FUNCTION_BLOCK FB_LGHeatpump implements IF_Heatpump
VAR_IN_OUT
	MBMaster		:	ModbusRtuMasterV2_KL6x22B;
END_VAR

VAR_OUTPUT
	Get				:	ST_HeatPump_Get;

END_VAR

VAR_IN_OUT CONSTANT
	st_params		: 	ST_Coolingsystem_params;
END_VAR

VAR_INPUT
	ACPowerStatus	:	BOOL;
	HeatPumpID		:	BYTE;
	SFCInit			:	BOOL;
	e_ID				:	eObject_ID := eObject_ID.HeatPump;
END_VAR
		
VAR
	ton_MBBUSYTimeOut		: TON := (PT := T#10s);
	DataBuffer				:	ARRAY[0..50] OF WORD;
	ton_modbusStuckTrigger	:	Ton	:=	(PT := T#5S);
	Ton_ErrorTimer			:	Ton := (PT := T#5M);
	MBRetryCount			:	BYTE;
	MBFree					:	BOOL;
	bMBActive				:	BOOL;
	ftrig_ModbusStartTrigger		:	f_Trig;
	TransmissionDoneTrigger	:	F_Trig;
	rtrig_ManualModbusStartTrigger : r_trig;
	btest	:	BOOL;
	ManADDR : BYTE;
	ton_testTimer	:	Ton := (Pt := T#100MS);
	TP_ModbusStartTriggerDelay	:	TP := (PT := TIME#50MS);
	u_counter				:	UINT;
END_VAR

VAR
	RequestedSetpoint				:	st_OperatingPoint;
	b_EMStop						:	BOOL;
	b_resetErrors					:	BOOL;
	t_RemainingPreheatingTime	:	TIME;
	sPressureErrorText			:	STRING;
	sCompressorErrorText		:	STRING;
	sPumpErrorText				:	STRING;
	sWaterTempErrorText			:	STRING;
END_VAR

VAR PERSISTENT
	dt_LastHPOperationTime	:	DT := DT#1970-1-1-0:0:0.000;
END_VAR


VAR
	CoilStatus		:	BYTE;
	LGget	:	LG_get;
	LGset	:	LG_SET;

	HeatpumpEMOperationAvailable	:	Bool;
END_VAR

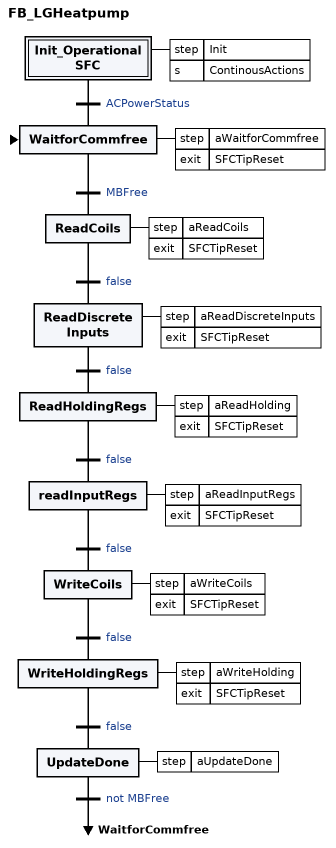
INITIAL_STEP Init_OperationalSFC:
    Init(N);  // step action
    ContinousActions(s);
END_STEP
TRANSITION FROM Init_OperationalSFC TO WaitforCommfree
    := ACPowerStatus;
END_TRANSITION
STEP WaitforCommfree:
    aWaitforCommfree(N);  // step action
    SFCTipReset(P0);  // exit action
END_STEP
TRANSITION FROM WaitforCommfree TO ReadCoils
    := MBFree;
END_TRANSITION
STEP ReadCoils:  // max time T#2S
    aReadCoils(N);  // step action
    SFCTipReset(P0);  // exit action
END_STEP
TRANSITION FROM ReadCoils TO ReadDiscreteInputs
    := false;
END_TRANSITION
STEP ReadDiscreteInputs:
    aReadDiscreteInputs(N);  // step action
    SFCTipReset(P0);  // exit action
END_STEP
TRANSITION FROM ReadDiscreteInputs TO ReadHoldingRegs
    := false;
END_TRANSITION
STEP ReadHoldingRegs:
    aReadHolding(N);  // step action
    SFCTipReset(P0);  // exit action
END_STEP
TRANSITION FROM ReadHoldingRegs TO readInputRegs
    := false;
END_TRANSITION
STEP readInputRegs:
    aReadInputRegs(N);  // step action
    SFCTipReset(P0);  // exit action
END_STEP
TRANSITION FROM readInputRegs TO WriteCoils
    := false;
END_TRANSITION
STEP WriteCoils:
    aWriteCoils(N);  // step action
    SFCTipReset(P0);  // exit action
END_STEP
TRANSITION FROM WriteCoils TO WriteHoldingRegs
    := false;
END_TRANSITION
STEP WriteHoldingRegs:
    aWriteHolding(N);  // step action
    SFCTipReset(P0);  // exit action
END_STEP
TRANSITION FROM WriteHoldingRegs TO UpdateDone
    := false;
END_TRANSITION
STEP UpdateDone:
    aUpdateDone(N);  // step action
END_STEP
TRANSITION FROM UpdateDone TO WaitforCommfree
    := not MBFree;
END_TRANSITION

METHOD AllowMBComm : BOOL
VAR_INPUT
	b_AllowComm	:	Bool;
END_VAR
MBFree	:= b_AllowComm;
END_METHOD

ACTION aReadCoils:
bMBActive := TRUE;

MBMaster.ReadCoils(	UnitID 		:= 	HeatPumpID,
					Quantity 	:= 	5,
					MBAddr		:=	0,				
					cbLength 	:= 	6,
					pMemoryAddr	:=	ADR(CoilStatus),
					Execute		:=	ftrig_ModbusStartTrigger.Q,
				);
	

IF TransmissionDoneTrigger.q THEN
	IF NOT MBMaster.Error THEN
		//Full datastruct for debug purposes. Can be removed later
		LGget.Coils.b_EnableOperation := CoilStatus.0;
		LGget.Coils.b_EnableSwwOperation := CoilStatus.1;
		LGget.Coils.b_EnableSilentMode := CoilStatus.2;
		LGget.Coils.b_EnableDesinfectionMode := Coilstatus.3;
		LGget.Coils.b_EmstopActive := CoilStatus.4;
		LGget.Coils.b_EnableEmStop := CoilStatus.5;
		//Full datastruct for debug purposes. Can be removed later
		
	ELSE
		MBRetryCount := MBRetryCount + 1;
	END_IF
	
	sfctip := TRUE;
END_IF


get.HeatpumpData.w_ErrorList[1] := lgget.Data.UI_ErrorCode;
get.Setpoint := lgget.Control.r_Setpoint1;
END_ACTION

ACTION aReadDiscreteInputs:


MBMaster.ReadInputStatus(	UnitID 		:= 	HeatPumpID,
							Quantity 	:= 	16,
							MBAddr		:=	0,
							cbLength 	:= 	SIZEOF(Databuffer),
							pMemoryAddr	:=	ADR(DataBuffer),
							Execute		:=	ftrig_ModbusStartTrigger.Q,
						);



IF TransmissionDoneTrigger.q THEN
	IF NOT MBMaster.Error THEN
		//Full datastruct for debug purposes. Can be removed later
		LGget.Status.b_WaterFlowNOK := DataBuffer[0].0;
		LGget.Status.b_WaterPumpOn := DataBuffer[0].1;
		LGget.Status.b_ExtWaterPumpOn := DataBuffer[0].2;
		LGget.Status.b_CompressorOn := DataBuffer[0].3;
		LGget.Status.b_DefrostOn := DataBuffer[0].4;
		LGget.Status.b_SWWModeOn := DataBuffer[0].5;
		LGget.Status.b_SWWTankDesinfectionActive := DataBuffer[0].6;
		LGget.Status.b_SilentModeOn := DataBuffer[0].7;
		LGget.Status.b_CoolingActive := DataBuffer[0].8;
		LGget.Status.b_SolarPumpActive := DataBuffer[0].9;
		LGget.Status.b_BackupHeater1Active := DataBuffer[0].10;
		LGget.Status.b_BackupHeater2Active := DataBuffer[0].11;
		LGget.Status.b_SWWBoostHeaterActive := DataBuffer[0].12;
		LGget.Status.b_ErrorActive := DataBuffer[0].13;
		LGget.Status.b_EMOperationAvailable := DataBuffer[0].14;
		LGget.Status.b_EMSWWOperationAvailable := DataBuffer[0].15;
		LGget.Status.b_MixPumpActive := DataBuffer[1].0;
		//Full datastruct for debug purposes. Can be removed later
		
		get.Events.b_PumpError := DataBuffer[0].0;
		get.HeatpumpData.b_DefrostingActive := DataBuffer[0].4;
		
		
		//error active and no em operation allowed
		IF DataBuffer[0].13 THEN
			get.HeatPumpState := eHeatpumpstate.ERROR;
			IF NOT DataBuffer[0].14 THEN
				HeatpumpEMOperationAvailable := FALSE;
			ELSE
				HeatpumpEMOperationAvailable := TRUE;
			END_IF
		ELSIF get.HeatPumpState = eHeatpumpstate.ERROR THEN
			get.HeatPumpState := eHeatpumpstate.Initializing;
			HeatpumpEMOperationAvailable := FALSE;
		END_IF
		
		//done, preset for next step
		MBRetryCount := 0;
	ELSE
		MBRetryCount := MBRetryCount + 1;
	END_IF
	sfctip := TRUE;
END_IF
END_ACTION

ACTION aReadHolding:

MBMaster.ReadRegs(	UnitID 		:= 	HeatPumpID,
					Quantity 	:= 	10,
					MBAddr		:=	0,
					cbLength 	:= 	SIZEOF(Databuffer),
					pMemoryAddr	:=	ADR(DataBuffer),
					Execute		:=	ftrig_ModbusStartTrigger.Q,
					);


IF TransmissionDoneTrigger.q THEN
	IF NOT MBMaster.Error THEN
		LGget.Control.ui_OperatingMode := Databuffer[0];
		LGget.Control.ui_ControlMode := Databuffer[1];
		LGget.Control.r_Setpoint1 := (WORD_TO_REAL(Databuffer[2])/10);
		LGget.Control.r_RoomSetpoint := (WORD_TO_REAL(Databuffer[3])/10);
		LGget.Control.ui_TempShiftValue := Databuffer[4];
		LGget.Control.r_Setpoint2 := (WORD_TO_REAL(Databuffer[5])/10);
		LGget.Control.r_RoomSetpoint2 := (WORD_TO_REAL(Databuffer[6])/10);
		LGget.Control.ui_TempShiftValue2 := Databuffer[7];
		LGget.Control.r_DHWgoalTemp := (WORD_TO_REAL(Databuffer[8])/10);
		LGget.Control.ui_EnergyStatus := Databuffer[9];
		
		get.Setpoint := (WORD_TO_REAL(Databuffer[2])/10);


		IF get.HeatPumpState <> eHeatpumpstate.ERROR THEN
			CASE lgget.Data.ui_OperationalMode OF
				0:
					get.HeatPumpState := eHeatpumpstate.Standby;
				1:
					get.HeatPumpState := eHeatpumpstate.Active_Cooling;
				2:
					get.HeatPumpState := eHeatpumpstate.Active_Heating;
			END_CASE
		END_IF
	
		//done, preset for next step
		MBRetryCount := 0;

	ELSE
		MBRetryCount := MBRetryCount + 1;
		
	END_IF
	sfctip := TRUE;
END_IF
END_ACTION

ACTION aReadInputRegs:
//SFCTip := FALSE;

MBMaster.ReadInputRegs ( 
					UnitID 		:= 	HeatPumpID,
					Quantity 	:= 	13,
					MBAddr		:=	0,
					cbLength 	:= 	SIZEOF(Databuffer),
					pMemoryAddr	:=	ADR(Databuffer),
					Execute		:=	ftrig_ModbusStartTrigger.Q,		
					);
				
IF TransmissionDoneTrigger.q THEN
	IF NOT MBMaster.Error THEN
		
	//Full datastruct for debug purposes. Can be removed later
		LGget.Data.UI_ErrorCode := Databuffer[0];	
		LGget.Data.ui_OperationalMode := (Databuffer[1]);	
		LGget.Data.r_CoolantInletTemp := WORD_TO_REAL((Databuffer[2]))/10;	
		LGget.Data.r_CoolantOutletTemp := WORD_TO_REAL((Databuffer[3]))/10;
		LGget.Data.r_BackupHeaterTemp := WORD_TO_REAL((Databuffer[4]))/10;
		LGget.Data.r_SWWTankTemp :=  WORD_TO_REAL((Databuffer[5]))/10;
		LGget.Data.r_SolarCollectorTemp := WORD_TO_REAL((Databuffer[6]))/10;
		LGget.Data.r_RoomTemp1 := WORD_TO_REAL((Databuffer[7]))/10;
		LGget.Data.r_FlowRate := WORD_TO_REAL((Databuffer[8]))/10;
		LGget.Data.r_FlowTempCircuit2 := WORD_TO_REAL((Databuffer[9]))/10;
		LGget.Data.r_RoomTemp2 := WORD_TO_REAL((Databuffer[10]))/10;
		LGget.Data.UI_EnergyStatus := (Databuffer[11]);
		LGget.Data.r_OutsideTemp := WORD_TO_REAL((Databuffer[12]))/10;
	//full datastruct for debug purposes. can be removed later	
		
		
		get.HeatpumpData.w_ErrorList[1] := Databuffer[0];
		Get.HeatpumpData.r_InletWaterTemp := WORD_TO_REAL((Databuffer[2]))/10;	
		get.HeatpumpData.r_OutletWaterTemp := WORD_TO_REAL((Databuffer[3]))/10;
		get.HeatpumpData.r_OutdoorTemp := WORD_TO_REAL((Databuffer[12]))/10;
		get.HeatpumpData.ui_WaterFlowRate := TO_UINT(Databuffer[8]/10);
	ELSE
		MBRetryCount := MBRetryCount + 1;
	END_IF
	sfctip := TRUE;
END_IF
END_ACTION

ACTION aUpdateDone:
SFCTip := FALSE;
bMBActive := FALSE;
END_ACTION

ACTION aWaitforCommfree:
//SFCTip := FALSE;
//b_EnableTransmission	:= FALSE;
//ModbusStartTrigger(clk := b_EnableTransmission);
END_ACTION

ACTION aWriteCoils:


CoilStatus.0 := requestedSetpoint.OperatingMode <> eHeatpumpMode.Standby; // operation off

CoilStatus.5 := EMHeatingModeRequired();


//IF get.HeatPumpState = eHeatpumpState.Initializing THEN
	MBMaster.WriteMultipleCoils(	UnitID 		:= 	HeatPumpID,
									Quantity 	:= 	5,
									MBAddr		:=	0,
									cbLength 	:= 	1,
									pMemoryAddr	:=	ADR(CoilStatus),
									Execute		:=	ftrig_ModbusStartTrigger.Q,	
						);
	
	IF TransmissionDoneTrigger.q THEN
		IF NOT MBMaster.Error THEN
			sfctip := TRUE;
			
		ELSE
			MBRetryCount := MBRetryCount + 1;
			sfctip := NOT sfctip;
		END_IF
	END_IF
//ELSE
//	sfctip := NOT sfctip;
//END_IF
END_ACTION

ACTION aWriteHolding:

CASE requestedSetpoint.OperatingMode OF
	eHeatpumpMode.Cooling:
		Databuffer[0] := 0; // cooling mode
		Databuffer[2] := REAL_TO_WORD(requestedSetpoint.Setpoint*10);
	eHeatpumpMode.Heating:
		Databuffer[0] := 4; // Heating mode
		Databuffer[2] := REAL_TO_WORD(requestedSetpoint.Setpoint*10);	
END_CASE
		
Databuffer[1] := 1; // inlet temperature control
Databuffer[3] := 0;
Databuffer[4] := 0;
Databuffer[5] := 0;
Databuffer[6] := 0;
Databuffer[7] := 0;
Databuffer[8] := 0;
Databuffer[9] := 2; // normal operation

MBMaster.WriteRegs (
		UnitID 		:= 	HeatPumpID,
		Quantity 	:= 	10,
		MBAddr		:=	0,
		cbLength 	:= 	SIZEOF(Databuffer),
		pMemoryAddr	:=	ADR(Databuffer),
		Execute		:=	ftrig_ModbusStartTrigger.Q,		
);



IF TransmissionDoneTrigger.q THEN
	IF NOT MBMaster.Error THEN
		//done, preset for next step

		MBRetryCount := 0;;
	ELSE
		MBRetryCount := MBRetryCount + 1;
	END_IF
	sfctip := TRUE;
END_IF
END_ACTION

ACTION ContinousActions:
//sfctip := False;
ton_modbusStuckTrigger(in := NOT ton_modbusStuckTrigger.q AND NOT TP_ModbusStartTriggerDelay.q);
TP_ModbusStartTriggerDelay(IN := NOT MBMaster.BUSY AND NOT ton_modbusStuckTrigger.q );
ftrig_ModbusStartTrigger(clk := TP_ModbusStartTriggerDelay.Q);

IF SFCError THEN
	SFCError := FALSE;
	get.Events.b_CommWarning := TRUE;
END_IF

IF NOT ACPowerStatus THEN
	IF get.HeatPumpState <> eHeatpumpstate.OFF THEN
		SFCReset := TRUE;
	END_IF
ELSIF get.HeatPumpState = eHeatpumpState.OFF THEN
	get.HeatPumpState := eHeatpumpState.Initializing;
END_IF

//safeguard, should the sfc get stuck, heatpumpsystem can revoke MB rights and SFC resets.
//IF NOT MBfree AND bMBActive AND NOT MBMaster.BUSY THEN
//	SFCReset := TRUE;
//END_IF 



HeatpumpPreheatControl();


//reset mb master if stuck in busy
ton_MBBUSYTimeOut(IN := MBmaster.BUSY);
IF ton_MBBUSYTimeOut.Q THEN
	MBMaster.ReadCoils();
	MBMaster.ReadInputStatus();
	MBMaster.ReadRegs();
	MBMaster.WriteMultipleCoils();
	MBMaster.WriteRegs();
	MBMaster.WriteSingleRegister();
END_IF

//Reset heatpump when error occurs, but after a bit of cooldown time.
//Maybe add a functionality to stop trying after x tries to prevent continuous reset cycles
Ton_ErrorTimer(in := get.Events.b_CompressorError OR 
					get.Events.b_FanError OR 
					get.Events.b_PressureError OR 
					get.Events.b_WaterTempError OR 
					get.Events.b_PumpError );
IF Ton_ErrorTimer.Q THEN
	b_resetErrors := TRUE;
END_IF

TransmissionDoneTrigger(clk := MBMaster.Busy);
MBMaster.Timeout		:= st_params.t_ModbusTimeOut;		

get.Events.b_CommWarning := MBRetryCount > st_params.i_modbusRetries;

IF TRUE THEN
	CASE requestedSetpoint.OperatingMode OF
		eHeatPumpMode.Standby:
			LGset.Coils.b_EnableOperation := FALSE;
			LGset.Regs.ui_OperatingMode := 3;
		eHeatPumpMode.Cooling:
			LGset.Coils.b_EnableOperation := TRUE;
			LGset.Regs.r_Setpoint1 := RequestedSetpoint.Setpoint;
			LGset.Regs.ui_OperatingMode := 0;
		eHeatPumpMode.Heating:
			LGset.Coils.b_EnableOperation := TRUE;
			LGset.Regs.r_Setpoint1 := RequestedSetpoint.Setpoint;
			LGset.Regs.ui_OperatingMode := 4;
	END_CASE
END_IF
END_ACTION

METHOD EMHeatingModeRequired : BOOL
VAR_INPUT
END_VAR
//some heatpump faults allow for emergency heating operation. If this occurs and heating is required, switch to emergency heating mode to keep the system warm.
//Cooling operation is not available in this mode.

IF lgget.Status.b_EMOperationAvailable AND RequestedSetpoint.OperatingMode = eHeatpumpmode.Heating THEN
	EMHeatingModeRequired := TRUE;
ELSE
	EMHeatingModeRequired := FALSE;
END_IF
END_METHOD

METHOD EMStop : BOOL
RequestedSetpoint.OperatingMode := eHeatpumpMode.Standby;
b_Emstop := TRUE;
EMstop := TRUE;
END_METHOD

METHOD GetDiagnostics 
VAR_IN_OUT
	AddError		: ARRAY [*] OF FB_AddErrorST;
	a_ActiveEvents	: ARRAY [*] OF ST_ErrorStruct;
	w_Index			: WORD;
END_VAR

VAR_OUTPUT
	b_errorActive	: BOOL;
	b_warningActive	: BOOL;
END_VAR

VAR
	by_errCt	: BYTE;
	by_warnCt	: BYTE;
	HPErrorText	: STRING;
END_VAR
	(*Modbus comm fault*)	AddError[w_Index](
			b_ErrorTrig			:= Get.Events.b_commwarning,
			out_ST_Error			:= a_ActiveEvents[w_Index],
			w_ErrorID				:= 30 + ((HeatPumpID-1)*10),
			e_ObjectID				:= e_ID,
			s_Message				:= 'Modbus communication fault',
			e_sev					:= eSeverity.Warning,	
			b_AutoClear			:= TRUE,
			t_TriggerTime		:=	T#60s,
			//in_e_ErrAckAccess		:= TRUE,
			);
		w_Index := w_Index +1;
		
CASE get.HeatpumpData.w_ErrorList[1] OF
	0:										HPErrorText := '';
	1, 8, 13, 19, 44:						HPErrorText := 'Misc Sensor error';
	2, 6, 16, 17, 18, 41, 45, 46, 65, 114:	HPErrorText := 'Temperature sensor error';
	10:										HPErrorText := 'Water pump blocked';
	3, 5, 53, 52:							HPErrorText := 'Internal comm error';
	9, 60:									HPErrorText := 'Eeprom error';
	14:										HPErrorText := 'Flow error';
	15:										HPErrorText := 'Water outlet overheat';
	20:										HPErrorText := 'Heater thermal fuse failed';
	21, 22, 27, 29:							HPErrorText := 'Compressor overcurrent';
	26: 									HPErrorText := 'Compressor fault';
	32: 									HPErrorText := 'Compressor output overtemperature';
	23: 									HPErrorText := 'DC Voltage error';
	35: 									HPErrorText := 'Low pressure error';
	43:   									HPErrorText := 'pressure sensor error';
	54:   									HPErrorText := 'Input phase error';
	61:   									HPErrorText := 'condensor overtemperature error';
	62:   									HPErrorText := 'heatsink overtemperature error'; 
	67:  									HPErrorText := 'Fan blocked error';
ELSE
	HPErrorText := 'Unknown error';
END_CASE


		
	(*Heatpump fault*)	AddError[w_Index](
			b_ErrorTrig				:= get.HeatpumpData.w_ErrorList[1] <> 0,
			out_ST_Error			:= a_ActiveEvents[w_Index],
			w_ErrorID				:= 31 + ((HeatPumpID-1)*10),
			s_Message				:= concat(concat(concat('Heatpump fault: ', TO_STRING(get.HeatpumpData.w_ErrorList[1])), ' :'), HPErrorText),
			e_sev					:= eSeverity.Warning,	
			b_AutoClear				:= True,
			t_TriggerTime			:=	T#1S,
			//in_e_ErrAckAccess		:= TRUE,
			);
		w_Index := w_Index +1;
	
	
	(*Heatpump warning*)			AddError[w_Index](
			b_ErrorTrig			:= LGGet.Coils.b_EnableSwwOperation AND lgget.Status.b_EMOperationAvailable,
			out_ST_Error		:= a_ActiveEvents[w_Index],
			w_ErrorID			:= 32 + ((HeatPumpID-1)*10),
			s_Message			:= 'Emergency operation active, performance may be restricted',
			e_sev				:= eSeverity.Warning,	
			b_AutoClear			:= FALSE,
			t_TriggerTime		:=	T#1S,
			//in_e_ErrAckAccess		:= TRUE,
			);
		w_Index := w_Index +1;
		

//	(*Heatpump Pump fault*)			AddError[w_Index](
//			b_ErrorTrig			:= Get.Events.b_PumpError,
//			out_ST_Error			:= a_ActiveEvents[w_Index],
//			w_ErrorID				:= 33 + ((HeatPumpID-1)*10),
//			s_Message				:= 'pump fault',
//			e_sev					:= eSeverity.Warning,	
//			b_AutoClear			:= FALSE,
//			t_TriggerTime		:=	T#1S,
//			//in_e_ErrAckAccess		:= TRUE,
//			);
//		w_Index := w_Index +1;	
		
	(*Heatpump Preheating active*)			AddError[w_Index](
			b_ErrorTrig				:= Get.Events.b_HeatpumpPreheatingActive,
			out_ST_Error			:= a_ActiveEvents[w_Index],
			w_ErrorID				:= 34 + ((HeatPumpID-1)*10),
			s_Message				:= concat('Heatpump preheating active for ', TO_STRING(t_RemainingPreheatingTime)),
			e_sev					:= eSeverity.Info,	
			b_AutoClear				:= TRUE,
			);
		w_Index := w_Index +1;
END_METHOD

METHOD PRIVATE HeatpumpPreheatControl : BOOL
VAR
	b_PreheatingRequired	:	BOOL;
END_VAR

VAR_INST
	ton_PreheatingTimer	:	Ton;
END_VAR
//enable operation
ton_PreheatingTimer(IN:= ACPowerStatus, PT:= TO_TIME(st_params.dw_HeatpumpOperationDelay*1000*60));
b_PreheatingRequired := ((DT_TO_INT(GVL.dt_SystemDateTime) - DT_TO_INT(dt_LastHPOperationTime))/60) > st_params.i_SkipHPPreheatingTime;

t_RemainingPreheatingTime := ton_PreheatingTimer.PT - ton_preheatingTimer.ET;

IF ton_PreheatingTimer.Q THEN
	dt_LastHPOperationTime := GVL.dt_SystemDateTime;
	t_RemainingPreheatingTime := T#0ms;
END_IF

get.Events.b_HeatpumpPreheatingActive := b_PreheatingRequired AND ACPowerStatus ;
END_METHOD

ACTION Init:
get.HeatPumpState := eHeatpumpstate.OFF;
bmbActive := FALSE;
SFCReset := FALSE;
get.Events.b_CommWarning := FALSE;
MBRetryCount := 0;
END_ACTION

METHOD MBCommBusy : BOOL
VAR_INPUT
END_VAR
MBCommBusy := bMBActive;
END_METHOD

METHOD ParseHeatPumpErrors : BOOL
VAR_INPUT
	w_Alarms1	:	WORD;
	w_Alarms2	:	WORD;
	w_Alarms3	:	WORD;
	w_Alarms4	:	WORD;
	w_Alarms5	:	WORD;
	w_Alarms6	:	WORD;
	w_Alarms7	:	WORD;
END_VAR		


VAR_IN_OUT
	get	:	ST_HeatPump_Get;	
END_VAR




get.events.b_ProbeError		:=	WORD_TO_BOOL(w_Alarms3) OR WORD_TO_BOOL(w_Alarms4) OR w_Alarms5.0;

get.events.b_PressureError		:=	w_Alarms1.0 OR	//E001: High Pressure
									w_Alarms1.1 OR //E002: Low Pressure
									w_Alarms2.3;	//E020: Inverted Pressure Transducers
									
sPressureErrorText := '';
IF get.events.b_PressureError THEN
	sPressureErrorText := concat(sPressureErrorText, SEL(w_Alarms1.0, '', ' E001'));
	sPressureErrorText := concat(sPressureErrorText, SEL(w_Alarms1.1, '', ' E002'));
	sPressureErrorText := concat(sPressureErrorText, SEL(w_Alarms2.3, '', ' E020'));
END_IF
									
get.events.b_CompressorError	:=	w_Alarms1.2 OR //E003: Compressor overheated
									w_Alarms1.7 OR //E008: Compressor underspeed
									w_Alarms1.8 OR	//E009: High disch temp
									w_Alarms1.12 OR //E013: Comp2 Overheated
									w_Alarms2.2 OR	//E019: CP2 High disch temp
									w_Alarms2.6 OR	//E023: Comp3 Overheated
									w_Alarms5.1 OR //'E801: Link Inverter1',
									w_Alarms5.2 OR //'E802: Link Inverter2',
									w_Alarms5.3 OR //'E803: Link Inverter3',
									w_Alarms5.4 OR //'E851: HWfault Inverter1',
									w_Alarms5.5 OR //'E852: HWfault Inverter2',
									w_Alarms5.6 OR //'E853: HWfault Inverter3',
									w_Alarms5.7 OR //'E861: OverCurrent Inv1',
									w_Alarms5.8 OR //'E862: OverCurrent Inv2',
									w_Alarms5.9 OR //'E863: OverCurrent Inv3',
									w_Alarms5.10 OR //'E871: High Temp Inv1',
									w_Alarms5.11 OR //'E872: High Temp Inv2',
									w_Alarms5.12 OR //'E873: High Temp Inv3',
									w_Alarms5.13 OR //'E881: Bad Voltage Inv1',
									w_Alarms5.14 OR //'E882: Bad Voltage Inv2',
									w_Alarms5.15 OR //'E883: Bad Voltage Inv3',
									w_Alarms6.0 OR //E891: Phase Seq Inv1',
									w_Alarms6.1 OR //'E892: Phase Seq Inv2',
									w_Alarms6.2 OR //'E893: Phase Seq Inv3',
									w_Alarms6.3 OR //'E901: Model err Inv1',
									w_Alarms6.4 OR //'E902: Model err Inv2',
									w_Alarms6.5 OR //'E903: Model err Inv3',
									w_Alarms6.6 OR //'E911: Ovl error Inv1',
									w_Alarms6.7 OR //'E9112: Ovl error Inv2',
									w_Alarms6.8 OR //'E913: Ovl error Inv3',
									w_Alarms6.9 OR //'E921: Overc PFC Inv1',
									w_Alarms6.10 OR //'E922: Overc PFC Inv2',
									w_Alarms6.11 OR //'E923: Overc PFC Inv3',
									w_Alarms6.12 OR //'E931: Int Com ERR Inv1',
									w_Alarms6.13 OR //'E932: Int Com ERR Inv2',
									w_Alarms6.14 OR //'E933: Int Com ERR Inv3',
									w_Alarms6.15 OR //'E941: Fault PFC Inv1',
									w_Alarms7.0 OR //E942: Fault PFC Inv2
									w_Alarms7.1 OR //'E943: Fault PFC Inv3',
									w_Alarms7.2 OR //'E951: Probe error Inv1',
									w_Alarms7.3 OR //'E952: Probe error Inv2',
									w_Alarms7.4 OR //'E953: Probe error Inv3',
									w_Alarms7.5 OR //'E961: Abnormal Cond Inv1',
									w_Alarms7.6 OR //'E962: Abnormal Cond Inv2',
									w_Alarms7.7 OR //'E963: Abnormal Cond Inv3',
									w_Alarms7.8 OR //'E971: Inv1 Eeprom Error',
									w_Alarms7.9 OR //'E972: Inv2 Eeprom Error',
									w_Alarms7.10 OR //'E973: Inv3 Eeprom Error',
									w_Alarms7.11;	//E029: CP3 High disch temp

sCompressorErrorText := '';
IF get.events.b_CompressorError THEN
	sCompressorErrorText := concat(sCompressorErrorText, SEL(w_Alarms1.2, '', ' E003'));
	sCompressorErrorText := concat(sCompressorErrorText, SEL(w_Alarms1.7, '', ' E008'));
	sCompressorErrorText := concat(sCompressorErrorText, SEL(w_Alarms1.8, '', ' E009'));
	sCompressorErrorText := concat(sCompressorErrorText, SEL(w_Alarms1.12, '', ' E013'));
	sCompressorErrorText := concat(sCompressorErrorText, SEL(w_Alarms2.2, '', ' E019'));
	sCompressorErrorText := concat(sCompressorErrorText, SEL(w_Alarms2.6, '', ' E023'));
	sCompressorErrorText := concat(sCompressorErrorText, SEL(w_Alarms5.1, '', ' E801'));
	sCompressorErrorText := concat(sCompressorErrorText, SEL(w_Alarms5.2, '', ' E802'));
	sCompressorErrorText := concat(sCompressorErrorText, SEL(w_Alarms5.3, '', ' E803'));
	sCompressorErrorText := concat(sCompressorErrorText, SEL(w_Alarms5.4, '', ' E851'));
	sCompressorErrorText := concat(sCompressorErrorText, SEL(w_Alarms5.5, '', ' E852'));
	sCompressorErrorText := concat(sCompressorErrorText, SEL(w_Alarms5.6, '', ' E853'));
	sCompressorErrorText := concat(sCompressorErrorText, SEL(w_Alarms5.7, '', ' E861'));
	sCompressorErrorText := concat(sCompressorErrorText, SEL(w_Alarms5.8, '', ' E862'));
	sCompressorErrorText := concat(sCompressorErrorText, SEL(w_Alarms5.9, '', ' E863'));
	sCompressorErrorText := concat(sCompressorErrorText, SEL(w_Alarms5.10, '', ' E871'));
	sCompressorErrorText := concat(sCompressorErrorText, SEL(w_Alarms5.11, '', ' E872'));
	sCompressorErrorText := concat(sCompressorErrorText, SEL(w_Alarms5.12, '', ' E873'));
	sCompressorErrorText := concat(sCompressorErrorText, SEL(w_Alarms5.13, '', ' E881'));
	sCompressorErrorText := concat(sCompressorErrorText, SEL(w_Alarms5.14, '', ' E882'));
	sCompressorErrorText := concat(sCompressorErrorText, SEL(w_Alarms5.15, '', ' E883'));
	sCompressorErrorText := concat(sCompressorErrorText, SEL(w_Alarms6.0 , '', ' E891'));
	sCompressorErrorText := concat(sCompressorErrorText, SEL(w_Alarms6.1 , '', ' E892'));
	sCompressorErrorText := concat(sCompressorErrorText, SEL(w_Alarms6.2 , '', ' E893'));
	sCompressorErrorText := concat(sCompressorErrorText, SEL(w_Alarms6.3 , '', ' E901'));
	sCompressorErrorText := concat(sCompressorErrorText, SEL(w_Alarms6.4 , '', ' E902'));
	sCompressorErrorText := concat(sCompressorErrorText, SEL(w_Alarms6.5 , '', ' E903'));
	sCompressorErrorText := concat(sCompressorErrorText, SEL(w_Alarms6.6 , '', ' E911'));
	sCompressorErrorText := concat(sCompressorErrorText, SEL(w_Alarms6.7 , '', ' E912'));
	sCompressorErrorText := concat(sCompressorErrorText, SEL(w_Alarms6.8 , '', ' E913'));
	sCompressorErrorText := concat(sCompressorErrorText, SEL(w_Alarms6.9 , '', ' E921'));
	sCompressorErrorText := concat(sCompressorErrorText, SEL(w_Alarms6.10, '', ' E922'));
	sCompressorErrorText := concat(sCompressorErrorText, SEL(w_Alarms6.11, '', ' E923'));
	sCompressorErrorText := concat(sCompressorErrorText, SEL(w_Alarms6.12, '', ' E931'));
	sCompressorErrorText := concat(sCompressorErrorText, SEL(w_Alarms6.13, '', ' E932'));
	sCompressorErrorText := concat(sCompressorErrorText, SEL(w_Alarms6.14, '', ' E933'));
	sCompressorErrorText := concat(sCompressorErrorText, SEL(w_Alarms6.15, '', ' E941'));
	sCompressorErrorText := concat(sCompressorErrorText, SEL(w_Alarms7.0 , '', ' E942'));
	sCompressorErrorText := concat(sCompressorErrorText, SEL(w_Alarms7.1 , '', ' E943'));
	sCompressorErrorText := concat(sCompressorErrorText, SEL(w_Alarms7.2 , '', ' E951'));
	sCompressorErrorText := concat(sCompressorErrorText, SEL(w_Alarms7.3 , '', ' E952'));
	sCompressorErrorText := concat(sCompressorErrorText, SEL(w_Alarms7.4 , '', ' E953'));
	sCompressorErrorText := concat(sCompressorErrorText, SEL(w_Alarms7.5 , '', ' E961'));
	sCompressorErrorText := concat(sCompressorErrorText, SEL(w_Alarms7.6 , '', ' E962'));
	sCompressorErrorText := concat(sCompressorErrorText, SEL(w_Alarms7.7 , '', ' E963'));
	sCompressorErrorText := concat(sCompressorErrorText, SEL(w_Alarms7.8 , '', ' E971'));
	sCompressorErrorText := concat(sCompressorErrorText, SEL(w_Alarms7.9 , '', ' E972'));
	sCompressorErrorText := concat(sCompressorErrorText, SEL(w_Alarms7.10, '', ' E973'));
	sCompressorErrorText := concat(sCompressorErrorText, SEL(w_Alarms7.11, '', ' E029'));
END_IF
								
get.events.b_ValveError		:=		w_Alarms2.11; //E041: Incongruent temps;


get.events.b_FanError			:=	w_Alarms1.2 OR //E004: Fan Overheated	
									w_Alarms1.13 OR //E014: Fan2 Overheated 
									w_Alarms2.7;	//E024: Fan3 Overheated					

get.events.b_PumpError			:=	w_Alarms1.5 OR	 	//E006: Lack of flow
									w_Alarms1.15 OR 	//E016: Pump Overheated
									w_Alarms2.9;		//E026: Pump2 Overheated

sPumpErrorText := '';
IF get.events.b_PumpError THEN
	sPumpErrorText := concat(sPumpErrorText, SEL(w_Alarms1.5, '', ' E006'));
	sPumpErrorText := concat(sPumpErrorText, SEL(w_Alarms1.15, '', ' E016'));
	sPumpErrorText := concat(sPumpErrorText, SEL(w_Alarms2.9, '', ' E026'));		
END_IF						
									
get.events.b_WaterTempError		:=	w_Alarms2.1 OR	//E018: OverTemperature
									w_Alarms1.4;	//E005: Frost

sWaterTempErrorText := '';									
IF get.events.b_WaterTempError THEN
	sWaterTempErrorText := concat(sWaterTempErrorText, SEL(w_Alarms1.5, '', ' E018'));
	sWaterTempErrorText := concat(sWaterTempErrorText, SEL(w_Alarms1.15, '', ' E005'));	
END_IF		


									
get.events.b_IOError			:=	w_Alarms2.14 OR 	//E101: IOMod1 Disconnected
									w_Alarms2.15; 		//E102: IOMod2 Disconnected
END_METHOD

METHOD Reset : BOOL
//until restarting the heatpump we don't know if errors are gone. So clear them for now.

get.Events.b_CompressorError := FALSE;
get.Events.b_FanError := FALSE;
get.Events.b_IOError := FALSE;
get.Events.b_PressureError := FALSE;
get.Events.b_ProbeError := FALSE;
get.Events.b_PumpError := FALSE;
get.Events.b_ValveError := FALSE;
get.Events.b_WaterTempError := FALSE;
get.Events.b_CommWarning := FALSE;
b_Emstop := FALSE;

MBRetryCount := 0;
Reset := true;
END_METHOD

METHOD Setpoint : BOOL
VAR_INPUT
	OperatingMode	:	eHeatpumpMode	:= 	eHeatpumpMode.Standby;
	Temperature		: 	REAL			:=	18;
END_VAR
IF get.HeatPumpState >= eHeatpumpstate.Standby AND 
	NOT get.Events.b_HeatpumpPreheatingActive AND 
	NOT b_EMstop THEN
	RequestedSetpoint.Setpoint		:= Temperature;
	RequestedSetpoint.OperatingMode := OperatingMode;
ELSE
	RequestedSetpoint.OperatingMode := eHeatPumpMode.Standby;
	RequestedSetpoint.Setpoint		:= 18.0;
END_IF

get.Setpoint := RequestedSetpoint.Setpoint;
END_METHOD

ACTION SFCTipReset:
SFCTip := FALSE;
END_ACTION

METHOD VariableMapping : BOOL
VAR_INPUT
END_VAR
END_METHOD

END_FUNCTION_BLOCK

(* stored: Version 1.1.0.1, ProductVersion 3.1.4024.12
   POU FB_LGHeatpump: Id {f7d951ca-38b2-4caf-969c-0440a565acad}, SpecialFunc None
   Folder Private methods: Id {57dd2361-cd1e-4605-958a-0c4dfaef2ad6}
   Folder SFC: Id {bd61a0c0-f4b6-4181-a314-65c8532efd9e}
   Folder Structs: Id {ff3c4713-1401-470c-aa66-4f4354dfa9f1}
   Method AllowMBComm: Id {523c4199-41fb-47fd-a8e6-46416c0d753d}
   Action aReadCoils: Id {17d5d889-5dc6-4c18-9f7b-e3770639388a}
   Action aReadDiscreteInputs: Id {b03b78a7-7ef3-49a6-9b40-f138c46410b4}
   Action aReadHolding: Id {703128ea-fd61-4142-a532-854700cedc29}
   Action aReadInputRegs: Id {fbc4850c-089e-43b3-b8e9-931681c8e914}
   Action aUpdateDone: Id {a76d3193-ed30-4543-9e89-78c90c05a4f9}
   Action aWaitforCommfree: Id {f6c1c3e9-abfd-42a0-8163-eb1d8155f68a}
   Action aWriteCoils: Id {38369746-549b-4398-8f07-0a3714a9ed3e}
   Action aWriteHolding: Id {597916a9-67f6-47c0-8d7b-7d5cbbb1b966}
   Action ContinousActions: Id {15e5100f-d98a-4435-8f5d-9dbe9de18380}
   Method EMHeatingModeRequired: Id {dc74603f-70fb-446b-949c-90e5312c3a12}
   Method EMStop: Id {97968dc4-bbc7-4d8f-8918-cdcb970a3fed}
   Method getDiagnostics: Id {c98abc38-1041-4146-831a-17074b3bbc02}
   Method HeatpumpPreheatControl: Id {ed5d95af-376f-4d3d-b94f-9906af06fd92}
   Action Init: Id {aecb5d15-6925-4b03-9006-cf0e38122960}
   Method MBCommBusy: Id {5dc47226-096c-40ba-a966-5a07e7c115bd}
   Method ParseHeatPumpErrors: Id {e944767b-9e57-4729-87e4-a132c7c9854e}
   Method Reset: Id {a04d23d6-1609-4365-9d01-c83980dc9203}
   Method Setpoint: Id {2c9d58e2-7e73-4bce-9d3f-336c598c86a3}
   Action SFCTipReset: Id {b924af9f-c4e4-4780-b851-f49fe6d0416b}
   Method VariableMapping: Id {7c12eb72-3452-4966-a349-d6dc89444751} *)
